FUNCTION_BLOCK TMP_SYMLINKS (* Composite Function Block Type *)
  (* Standard: 61499-2 *)
  (* Version 0.0, 10/2/2026, template *)
  PACKAGE Hidryco.HidrycoLib;
END_FUNCTION_BLOCK
